{attribute 'TcGenerated'}
{attribute 'no-analysis'}
{attribute 'linkalways'}
// This function has been automatically generated from the project information.
VAR_GLOBAL CONSTANT
	{attribute 'const_non_replaced'}
	stLibVersion_Cognex_Camera : ST_LibVersion := (iMajor := 0, iMinor := 1, iBuild := 2, iRevision := 0, nFlags := 0, sVersion := '0.1.2');
END_VAR

(* stored: Version 1.1.0.1, ProductVersion 3.1.4024.10
   GVL Global_Version: Id {b0405b1a-ba4b-4419-84be-d6279eff9904} *)
